// TIA Portal V19 export
DATA_BLOCK "DB_ANLAGE"   // DB1
{ S7_Optimized_Access := 'FALSE' }
AUTHOR : MS
// stored: AutoNumber false
   VAR RETAIN
      BA : Struct   // Betriebsarten
         Not_Aus : Bool := FALSE;   // Not-Aus ist betätigt
         free0 : Bool := FALSE;   // sonst Anlage vom PC bedienen, nur bei BA-Schalter auf Auto
         free1 : Bool := FALSE;   // sonst Automatikbetrieb ist nicht freigegeben
         Tippbetrieb : Bool := FALSE;   // Tippbetrieb
         Handbetrieb : Bool := FALSE;   // Handbetrieb
         Automat_ein : Bool := FALSE;   // Automatikbetrieb möglich
         Automat_aus : Bool := FALSE;   // Automatikbetrieb nicht möglich
         Anlauf_Auto : Bool := FALSE;   // Anlauf Automatik für Scanvorgang WT-Positionen auf letzte Automatikposition
         Einfahr_Stop : Bool := FALSE;   // Stoppt die Einfahrt von WT in die Anlage(Feierabendprogramm)
         Mess_on : Bool := FALSE;   // Einmessung aktiv
         Taktwechsel : Bool := FALSE;   // Taktwechsel durchführen
         SIM_HISPEED : Bool := FALSE;   // * Simulation erfolgt mit doppelter Geschwindigkeit
         Simulation : Bool := FALSE;   // * Simulation eingeschaltet
         COM_RST : Bool := TRUE;   // Complete Restart
         FP_Automat_ein : Bool := FALSE;   // Flankenmerker positive Flanke Taste Automat ein
         newConfig : Bool := FALSE;   // neue Konfiguration (Daten neu verteilen)
      END_STRUCT;
      config : Struct   // Anlagenkonfiguration
         ANZ_FW : Int := 1;   // * Anzahl der Transportwagen in der Anlage
         ANZ_QT : Int := 0;   // * Anzahl der Quertransporte in der Anlage
         ANZ_Reihen : Int := 1;   // * Anzahl der Reihen in der Anlage
         ANZ_Pos : Int := 30;   // * Anzahl der Positionen
         ANZ_WT : Int := 12;   // * Anzahl der vorhandenen WT-Datenbausteine
         ANZ_POS_per_Cyc : Int := 6;   // * Anzahl der bearbeiteten Positionen pro Zyklus
         maxWT_loop : Int := 5;   // * im freien System Anzahl der Befehle der größten Technologieschleife
         Anz_Opt_Pos : Int := 0;   // * Anzahl der in die Optimierungsrechnung eingehenden Positionen
         Anz_GR : Int := 0;   // * Anzahl der Gleichrichter
         Anz_TR : Int := 0;   // * Anzahl der Temperaturregler
         Anz_DZ : Int := 2;   // * Anzahl der Dosierzähler
         Anz_DP : Int := 8;   // * Anzahl Dosierpumpen
         AnaEventInt : Int := 600;   // * Analogevent Intervall
         Taktzeit_typ : Int := 480;   // * typische Taktzeit für Expoberechnung in getakteten Positionen
         Transzeit_typ : Int := 60;   // * typische Zeit für einen Austauschvorgang
         Reihen_Cnfg : Struct
            EndePos_R1 : Int := 30;   // * Reihendefinition, letzte Position in Reihe 1 (immer niedriger als EndePos_R2)
            EndePos_R2 : Int := 0;   // * Reihendefinition, letzte Position in Reihe 2 (immer niedriger als EndePos_R3)
            EndePos_R3 : Int := 0;   // * Reihendefinition, letzte Position in Reihe 3 (immer niedriger als EndePos_R4)
            EndePos_R4 : Int := 0;   // * Reihendefinition, letzte Position in Reihe 4 (immer niedriger als EndePos_R5)
            EndePos_R5 : Int := 0;   // * Reihendefinition, letzte Position in Reihe 5
         END_STRUCT;
         akt_FW : Int := 0;
         Old_Hour_Event : Int := 0;
         PC_exist : Bool := 0;   // * PC-Daten schreiben (es existiert ein EventAbnehmer [FC7])
         Diag_exist : Bool := 0;   // * Diagrammdaten schreiben (Diagrammdaten werden am PC aufgezeichnet)
         Anl_getaktet : Bool := TRUE;   // * 0=Anlage fährt Auftragsorientiert 1=Anlage wird mit Ketten gesteuert
         HW_exist : Bool := TRUE;   // * Höhenwechsel in der Anlage vorhanden
         Pos_absolut : Bool := TRUE;   // * Positionsbestimmung absolut für OB100-Init-Pos (wirkt nicht mehr am FW)
         Opti_exist : Bool := FALSE;   // * Optimierung vorhanden
         AL_Einfahrt : Bool := FALSE;   // Ware aufgeben!!
         Al_Ausfahrt : Bool := FALSE;   // Beladestand räumen!!
         Weg_Zeit_aus : Bool := FALSE;   // * Weg-Zeit-Events nicht schreiben
         EntmFromOpt : Bool := FALSE;   // * Entmetallisierungs-WT werden von der Optimierung berechnet
         M_Q_Hupe : Bool := TRUE;
         HW_Auto_search : Bool := FALSE;   // * FW sucht automatisch nach einer möglichen Höhenwechselposition
         FP_Taste_Reset : Bool := FALSE;
         Time_from_PC : Bool := 0;   // * Zeit wird vom PC gestellt (keine autom. Sommerzeit)
         FP_Stop_Taktende : Bool := FALSE;   // Flankenmerker Stop bei Taktende erreicht
         Temp_MW_aktiv : Bool := 0;   // * Event mittlere Temperatur (Event 18) aktiv
         FP_Einrichten : Bool := FALSE;
         FP_Hand : Bool := TRUE;
         FP_Automatik : Bool := FALSE;
         FP_In_Quitt : Bool := FALSE;   // Flankenmerker Fehlerquittung
         Hub_absolut : Bool := FALSE;   // Hubsesorik Absolutgeber
         Battf : Bool := FALSE;   // Batteriefehler OB81 (Durch Hardwareschalter an SPS "BATT_INDIC") quittierbar
         RESET_STATUS : Bool := FALSE;   // Wiederanlaufmerker nach Reset
         WT_Typ_Afg : Bool := FALSE;   // * WT-Typ wird bei Aufgabe vergeben
         TypChckDetail : Bool := TRUE;   // * WT-Typ wird ohne Maske B#16#F0 geprüft
         QT_Trocken_chk : Bool := FALSE;   // * einschalten, wenn Prüfung auf bit "immer schnell"
         FB9_Takt : Bool := FALSE;   // * FB9 aufrufen obwohl Anlage getaktet
         Use_FB_Ana : Bool := 0;   // * 1=FB110 verwenden 0=klassische Analogwerterfassung FC110
         Check_Profibus : Bool := TRUE;   // * Profibusteilnehmer überwachen! OB86,OB100,DB203,FC203
         NormalB : Bool := FALSE;   // 0: 151 / 161 1: nur 151
         res6 : Bool := FALSE;
         ReqUmsTakt : Bool := FALSE;   // Anforderung Umschaltung auf getaktet
      END_STRUCT;
      IN : Struct   // Hardwareeingänge Anlage
         S_Not_Aus : Bool := FALSE;   // Not-Aus ok
         S_St_Spng : Bool := TRUE;   // Steuerspannung ein
         Quitt_Err : Bool := FALSE;   // Fehlerquittung
         Quitt_Hupe : Bool := FALSE;   // Hupenquittierung
         Reset : Bool := FALSE;   // Reset Anlagenschalter
         Reparatur : Bool := FALSE;   // Reparaturbetrieb
         Lamp_Test : Bool := FALSE;   // Lampentest
         BA_Tipp : Bool := FALSE;   // BA Umschalter Tipp
         BA_Hand : Bool := TRUE;   // BA Umschalter Hand
         BA_Auto : Bool := FALSE;   // BA Umschalter Auto
         Stop_Anlage : Bool := FALSE;   // Anlage hält am Takt- bzw. Schichtende an
         Automat_aus : Bool := FALSE;   // Taste Automatikbetrieb verbieten
         Automat_ein : Bool := FALSE;   // Taste Automatikbetrieb erlauben
         Quit_Err_Galva : Bool := FALSE;   // Fehlerquittung per Galva
         res4 : Bool := FALSE;
         UT_Req : Bool := FALSE;   // Anforderung Umlufttrockner
         ReqEventTakt : Bool := FALSE;   // Anforderung EventTakt
         GR_ok : Bool := FALSE;   // Rückmeldung Event erfolgt
         TR_ok : Bool := FALSE;   // Rückmeldung Event erfolgt
         pH_LF_ok : Bool := TRUE;   // Rückmeldung Event erfolgt
         DP_ok : Bool := FALSE;   // Rückmeldung Event erfolgt
         res11 : Bool := FALSE;
         res12 : Bool := FALSE;
         res13 : Bool := FALSE;
         PC_offline : Bool := FALSE;   // PC-Komunikation ist unterbrochen
         AMS_Restart : Bool := FALSE;   // alle anstehenden Fehler neu senden
         Watch_Profibus : Bool := FALSE;   // Profibusüberwachung eingeschaltet
         res17 : Bool := FALSE;
         res18 : Bool := FALSE;
         res19 : Bool := FALSE;
         res20 : Bool := FALSE;
         AMS_Reset : Bool := FALSE;   // AMS-Reset durchführen (Resetknopf während nicht Tipp)
      END_STRUCT;
      OUT : Struct   // Hardwareausgänge Anlage
         Stoerung_Opt : Bool := FALSE;
         Stoerung_Aku : Bool := FALSE;
         MD_Auto : Bool := FALSE;
         Fehler_Quitt : Bool := FALSE;
         res1 : Bool := FALSE;
         res2 : Bool := FALSE;
         res3 : Bool := FALSE;
         FW_QT_Auto : Bool := FALSE;   // mind. ein FW/QT hat seinen Automatikbefehl noch nicht beendet
         TW_abgelehnt : Bool := FALSE;   // Taktwechsel wurde abgelehnt (durch Fehlerquittung löschen)
         WT_in_Anlage : Bool := FALSE;
         res7 : Bool := FALSE;
         res8 : Bool := FALSE;
         res9 : Bool := FALSE;
         res10 : Bool := FALSE;
         res11 : Bool := FALSE;
         res12 : Bool := FALSE;
         res13 : Bool := FALSE;
         res14 : Bool := FALSE;
         res15 : Bool := FALSE;
         res16 : Bool := FALSE;
         res17 : Bool := FALSE;
         res18 : Bool := FALSE;
         res19 : Bool := FALSE;
         res20 : Bool := FALSE;
         AnzUT_Req : Byte := 16#00;   // Anzahl der UT Anforderungen
      END_STRUCT;
      config2 : Struct
         Anzahl_HW : Int := 1;   // * Anzahl Höhenwechsel (Definition im DB53)
         Woscha_DB_1 : Int := 8;   // Datenbaustein für Wochenschaltuhr 1
         Woscha_DB_2 : Int := 0;   // Datenbaustein für Wochenschaltuhr 2
         Woscha_DB_3 : Int := 0;   // Datenbaustein für Wochenschaltuhr 3
         Woscha_DB_4 : Int := 0;   // Datenbaustein für Wochenschaltuhr 4
         resW4 : Int := 0;
         Anlagentakte : Int := 3;   // Anzahl Takte, welche WT durch die Anlage läuft
         resW6 : Int := 0;
         resW7 : Int := 0;
         resW8 : Int := 0;
         resW9 : Int := 0;
         resW10 : Int := 0;
         resW11 : Int := 0;
         resW12 : Int := 0;
         resW13 : Int := 0;
         resW14 : Int := 0;
         resW15 : Int := 0;
         resW16 : Int := 0;
         resW17 : Int := 0;
         resW18 : Int := 0;
         resW19 : Int := 0;
      END_STRUCT;
      FW1 : Struct
         FW_min : Int := 1;   // * FW Bereich min
         FW_max : Int := 30;   // * FW Bereich max
         RefPos : Int := 0;   // * Referenzposition (bei Absolutpositionierung 0)
         T_Nr : Int := 10;   // * Timer1
         resW : Int := 0;
      END_STRUCT;
      FW2 : Struct
         FW_min : Int := 0;   // * FW Bereich min
         FW_max : Int := 0;   // * FW Bereich max
         RefPos : Int := 0;   // * Referenzposition (bei Absolutpositionierung 0)
         T_Nr : Int := 0;   // * Timer1
         resW : Int := 0;
      END_STRUCT;
      FW3 : Struct
         FW_min : Int := 0;   // * FW Bereich min
         FW_max : Int := 0;   // * FW Bereich max
         RefPos : Int := 0;   // * Referenzposition (bei Absolutpositionierung 0)
         T_Nr : Int := 0;   // * Timer1
         resW : Int := 0;
      END_STRUCT;
      FW4 : Struct
         FW_min : Int := 0;   // * FW Bereich min
         FW_max : Int := 0;   // * FW Bereich max
         RefPos : Int := 0;   // * Referenzposition (bei Absolutpositionierung 0)
         T_Nr : Int := 0;   // * Timer1
         resW : Int := 0;
      END_STRUCT;
      FW5 : Struct
         FW_min : Int := 0;   // * FW Bereich min
         FW_max : Int := 0;   // * FW Bereich max
         RefPos : Int := 0;   // * Referenzposition (bei Absolutpositionierung 0)
         T_Nr : Int := 0;   // * Timer1
         resW : Int := 0;
      END_STRUCT;
      FW6 : Struct
         FW_min : Int := 0;   // * FW Bereich min
         FW_max : Int := 0;   // * FW Bereich max
         RefPos : Int := 0;   // * Referenzposition (bei Absolutpositionierung 0)
         T_Nr : Int := 0;   // * Timer1
         resW : Int := 0;
      END_STRUCT;
      FW7 : Struct
         FW_min : Int := 0;   // * FW Bereich min
         FW_max : Int := 0;   // * FW Bereich max
         RefPos : Int := 0;   // * Referenzposition (bei Absolutpositionierung 0)
         T_Nr : Int := 0;   // * Timer1
         resW : Int := 0;
      END_STRUCT;
      FW8 : Struct
         FW_min : Int := 0;   // * FW Bereich min
         FW_max : Int := 0;   // * FW Bereich max
         RefPos : Int := 0;   // * Referenzposition (bei Absolutpositionierung 0)
         T_Nr : Int := 0;   // * Timer1
         resW : Int := 0;
      END_STRUCT;
      FW9 : Struct
         FW_min : Int := 0;   // * FW Bereich min
         FW_max : Int := 0;   // * FW Bereich max
         RefPos : Int := 0;   // * Referenzposition (bei Absolutpositionierung 0)
         T_Nr : Int := 0;   // * Timer1
         resW : Int := 0;
      END_STRUCT;
      FW10 : Struct
         FW_min : Int := 0;   // * FW Bereich min
         FW_max : Int := 0;   // * FW Bereich max
         RefPos : Int := 0;   // * Referenzposition (bei Absolutpositionierung 0)
         T_Nr : Int := 0;   // * Timer1
         resW : Int := 0;
      END_STRUCT;
      FW11 : Struct
         FW_min : Int := 0;   // * FW Bereich min
         FW_max : Int := 0;   // * FW Bereich max
         RefPos : Int := 0;   // * Referenzposition (bei Absolutpositionierung 0)
         T_Nr : Int := 0;   // * Timer1
         resW : Int := 0;
      END_STRUCT;
      FW12 : Struct
         FW_min : Int := 0;   // * FW Bereich min
         FW_max : Int := 0;   // * FW Bereich max
         RefPos : Int := 0;   // * Referenzposition (bei Absolutpositionierung 0)
         T_Nr : Int := 0;   // * Timer1
         resW : Int := 0;
      END_STRUCT;
      FW13 : Struct
         FW_min : Int := 0;   // * FW Bereich min
         FW_max : Int := 0;   // * FW Bereich max
         RefPos : Int := 0;   // * Referenzposition (bei Absolutpositionierung 0)
         T_Nr : Int := 0;   // * Timer1
         resW : Int := 0;
      END_STRUCT;
      FW14 : Struct
         FW_min : Int := 0;   // * FW Bereich min
         FW_max : Int := 0;   // * FW Bereich max
         RefPos : Int := 0;   // * Referenzposition (bei Absolutpositionierung 0)
         T_Nr : Int := 0;   // * Timer1
         resW : Int := 0;
      END_STRUCT;
      FW15 : Struct
         FW_min : Int := 0;   // * FW Bereich min
         FW_max : Int := 0;   // * FW Bereich max
         RefPos : Int := 0;   // * Referenzposition (bei Absolutpositionierung 0)
         T_Nr : Int := 0;   // * Timer1
         resW : Int := 0;
      END_STRUCT;
      QT1 : Struct
         PosR1 : Byte := 16#00;   // * QT-Reihe1: Positionsnummer der ersten QT-Pos (bei Rückwärtsfahrt letzte Pos)
         PosR2 : Byte := 16#00;   // * QT-Reihe2: Positionsnummer der zweiten QT-Pos
         PosR3 : Byte := 16#00;   // * QT-Reihe3: Positionsnummer der dritten QT-Pos
         PosR4 : Byte := 16#00;   // * QT-Reihe4: Positionsnummer der vierten QT-Pos
         PosR5 : Byte := 16#00;   // * QT-Reihe5: Positionsnummer der fünften QT-Pos
         RefReihe : Byte := 16#00;   // * Referenzreihe nur angeben wenn mitfahrende Sensoren!!
         T_Nr : Int := 0;   // * Timer1
         Ketten_DB : Int := 0;   // * Eintrag == 0 --> QT besitzt keine Kette
      END_STRUCT;
      QT2 : Struct
         PosR1 : Byte := 16#00;   // * QT-Reihe1: Positionsnummer der ersten QT-Pos (bei Rückwärtsfahrt letzte Pos)
         PosR2 : Byte := 16#00;   // * QT-Reihe2: Positionsnummer der zweiten QT-Pos
         PosR3 : Byte := 16#00;   // * QT-Reihe3: Positionsnummer der dritten QT-Pos
         PosR4 : Byte := 16#00;   // * QT-Reihe4: Positionsnummer der vierten QT-Pos
         PosR5 : Byte := 16#00;   // * QT-Reihe5: Positionsnummer der fünften QT-Pos
         RefReihe : Byte := 16#00;   // * Referenzreihe nur angeben wenn mitfahrende Sensoren!!
         T_Nr : Int := 0;   // * Timer1
         Ketten_DB : Int := 0;   // * Eintrag == 0 --> QT besitzt keine Kette
      END_STRUCT;
      QT3 : Struct
         PosR1 : Byte := 16#00;   // * QT-Reihe1: Positionsnummer der ersten QT-Pos (bei Rückwärtsfahrt letzte Pos)
         PosR2 : Byte := 16#00;   // * QT-Reihe2: Positionsnummer der zweiten QT-Pos
         PosR3 : Byte := 16#00;   // * QT-Reihe3: Positionsnummer der dritten QT-Pos
         PosR4 : Byte := 16#00;   // * QT-Reihe4: Positionsnummer der vierten QT-Pos
         PosR5 : Byte := 16#00;   // * QT-Reihe5: Positionsnummer der fünften QT-Pos
         RefReihe : Byte := 16#00;   // * Referenzreihe nur angeben wenn mitfahrende Sensoren!!
         T_Nr : Int := 0;   // * Timer1
         Ketten_DB : Int := 0;   // * Eintrag == 0 --> QT besitzt keine Kette
      END_STRUCT;
      QT4 : Struct
         PosR1 : Byte := 16#00;   // * QT-Reihe1: Positionsnummer der ersten QT-Pos (bei Rückwärtsfahrt letzte Pos)
         PosR2 : Byte := 16#00;   // * QT-Reihe2: Positionsnummer der zweiten QT-Pos
         PosR3 : Byte := 16#00;   // * QT-Reihe3: Positionsnummer der dritten QT-Pos
         PosR4 : Byte := 16#00;   // * QT-Reihe4: Positionsnummer der vierten QT-Pos
         PosR5 : Byte := 16#00;   // * QT-Reihe5: Positionsnummer der fünften QT-Pos
         RefReihe : Byte := 16#00;   // * Referenzreihe nur angeben wenn mitfahrende Sensoren!!
         T_Nr : Int := 0;   // * Timer1
         Ketten_DB : Int := 0;   // * Eintrag == 0 --> QT besitzt keine Kette
      END_STRUCT;
      QT5 : Struct
         PosR1 : Byte := 16#00;   // * QT-Reihe1: Positionsnummer der ersten QT-Pos (bei Rückwärtsfahrt letzte Pos)
         PosR2 : Byte := 16#00;   // * QT-Reihe2: Positionsnummer der zweiten QT-Pos
         PosR3 : Byte := 16#00;   // * QT-Reihe3: Positionsnummer der dritten QT-Pos
         PosR4 : Byte := 16#00;   // * QT-Reihe4: Positionsnummer der vierten QT-Pos
         PosR5 : Byte := 16#00;   // * QT-Reihe5: Positionsnummer der fünften QT-Pos
         RefReihe : Byte := 16#00;   // * Referenzreihe nur angeben wenn mitfahrende Sensoren!!
         T_Nr : Int := 0;   // * Timer1
         Ketten_DB : Int := 0;   // * Eintrag == 0 --> QT besitzt keine Kette
      END_STRUCT;
   END_VAR
BEGIN
END_DATA_BLOCK
